TYPE T_CodePO : STRING[20];
END_TYPE

(* stored: Version 1.1.0.1
   DUT T_CodePO: Id {ac8a1938-32b4-4e9b-983a-c9c393136188} *)
